// TIA Portal V19 export
TYPE "TAx_Alarms"
// stored: Access Published
   STRUCT
      TOAxis : Bool;   // Alarm in technology object
      MCFunction : Bool;   // Alarm of MC function
      Drive : Bool;   // Alarm in the drive
      LimitMinus : Bool;   // Limit minus SW or HW reached
      LimitPlus : Bool;   // Limit plus SW or HW reached
   END_STRUCT;
END_TYPE
